{attribute 'GeneratedUsingTerminal: EK1122-0000-0018'}
{attribute addProperty BoxType "EK1122-0000-0018"}
{attribute addProperty Id "Beckhoff_EL4xxxsub_EK1100EK1100_AB5A94672"}
{attribute addProperty CRC "3389342480"}
{attribute addProperty Size "2"}
TYPE Beckhoff_EL4xxxEK1122_CA054310 EXTENDS EK1122_AB5A9467 :
STRUCT
	{attribute addProperty Name "Beckhoff_EL4xxxsub_EK1100"}
	{attribute addProperty PreviousPort "Beckhoff EL4xxxEK1122 : D"}
	Beckhoff_EL4xxxsub_EK1100 : EK1100_AB5A9467;
END_STRUCT
END_TYPE

(* stored: Version 1.2.0.0, ProductVersion 3.1.4024.9
   DUT Beckhoff_EL4xxxEK1122_CA054310: Id {2a811fda-30c0-41c6-aad0-7c07fb8ee97f} *)
